(* IEC 61131-3 sources: std_i2980_v2.06_cp053/Source/IMM/ieccontrol/ServiceNet, 6 files *)

(* ---- FBSendData.pu ---- *)
(*
@h    ! WARNING !
@h    The Kemro K2 system (including software) only meets category B according to EN 954-1,
@h    thus it is not intended for usage in safety-relevant control applications in the field
@h    of personal safety (e.g. emergency stop).
@h    To implement potentially necessary safety-relevant control tasks, always use additional
@h    external safety devices that are intended for the particular purpose, and meet the necessary
@h    functional safety.
@h    For further information see EN 954-1 (EN ISO 13849-1) and/or the K2-x00 user manual, chapter
@h    "CE conformity, directives and standards".

function block for sending data according to ServiceNet protocol to ServiceNet Server.
sends connection data and connection status on raising edge on execute
sends connection status information if status changed, but at least once each 30 seconds (keep alive).

ATTENTION: when changing content of send buffer:
-> ensure that maximum length does not exceed 255 characters per buffer element when concating strings,
   otherwise characters are truncated which will lead to an invalid object beeing sent.
-> ensure to CONCAT sClear String (255 x blank) at the end of each buffer-array element
   (to delete string data stored previously on that buffer element in case the new string is shorter)
-> a string data element started in a buffer element (character ") must be closed in the same buffer element
   because at the end of each 255 character buffer element a zero byte (string terminator) is inserted automatically.
   a zero byte is not allowed in string elements!
   therefore the maximum length of a string that can be sent is 255 - 2 = 253 characters.
*)

IMPORT_OVER_LISTFILE
 GET_RUNTIME
, ABVersionManager
, tyRequestFrom
, tsMachineInfo
, tnConnectionStatus
, tySBuf
, KNETWORK_TcpSend
, TON

END_IMPORT

FUNCTION_BLOCK FBSendData #DUMMY_EDIT_BLOCK

VAR_INPUT
 Execute : BOOL (* sends all data on raising edge, when TRUE: connection status is sent on valuechange and after 30 seconds elapsed without valuechange *);
 TcpHdl : REFERENCE (* handle of an established TCP connection to use for sending data *);
 VersionServiceNetClient : DINT (* ServiceNet protocol version used by client *);
END_VAR

VAR_IN_OUT
 abVersionInfo : ABVersionManager (* block for reading versioninfos and systemname *);
END_VAR

VAR_OUTPUT
 Error : BOOL (* indicates a send error *);
END_VAR

SYSTEM_VAR
 sv_RequestFrom : tyRequestFrom;
 sv_sTextMessage : STRING(255);
 sv_iRequestFromIdx : DINT;
 sv_iCpuId : LINT;
 sv_MachineInformation : tsMachineInfo;
 sv_ConnectionStatus : tnConnectionStatus;
 sv_iRemoteVisType : DINT;
END_VAR

VAR
 Buf : tySBuf (* send buffer *);
 fbTCPSend : KNETWORK_TcpSend (* block for sending data  *);
 bSendConnectionData : BOOL (* indicates all data should be sent *);
 bSendStatusOnly : BOOL (* indicates only status should be sent *);
 bExecuteOld : BOOL (* flag stores Execute state in previous cycle for detecting edges *);
 ts : TIME (* debug: timestamp start *);
 td : TIME (* debug: duration *);
 fbTonKeepAlive : TON (* keep alive timer *);
 iConnectionState : DINT (* integer value of sv_ConnectionState *);
 connectionStatusOld : tnConnectionStatus (* connection state in previous cycle - to detect state changed *);
 iSendBytes : UDINT (* number of bytes to send *);
 sByteLen : STRING(16) (* length information about data object to be sent to ServiceNet server *);
 sTmpString : STRING(63) (* helper string  *);
 sKVSVersion : STRING(63);
END_VAR

VAR CONSTANT
 sClear : STRING(255) := '                                                                                                                                                                                                                                                               ' (* string with 255 blanks (0x20) *);
END_VAR
#BEGIN_EDIT_BLOCK
(**************************************** WARNING ********************************************
 *** The KEBA Kemro K2 System including software is not intended for safety control tasks! ***
 ***                       For further information see Comment tab!                        ***
 *********************************************************************************************)

// keep alive message timer, start on raising edge of Execute input
fbTonKeepAlive(Execute, T#30s);

// data to send if keep alive timer elapsed or connection status changed
bSendStatusOnly := fbTonKeepAlive.Q OR (sv_ConnectionStatus <> connectionStatusOld);

// initialize TCP send block on raising edge
IF (Execute AND (NOT bExecuteOld)) THEN
    fbTCPSend(Execute := FALSE, TcpHdl := TcpHdl);
END_IF;

IF (Execute) THEN
   // send all connection data on raising edget of Execute flag
   bSendConnectionData := (NOT bExecuteOld);

   // send data?
   IF (bSendStatusOnly OR bSendConnectionData) THEN
       // reset keep alive timer
       fbTonKeepAlive(IN := FALSE);

       // timestamp for performance measurement
       ts := GET_RUNTIME();

       connectionStatusOld := sv_ConnectionStatus;

       // connection status to integer
       CASE (connectionStatusOld) OF
            nDisconnected:
                iConnectionState := 0;

            nConnecting:
                iConnectionState := 1;

            nRequestPending:
                iConnectionState := 2;

            nServiceAccepted:
                iConnectionState := 3;

            nServiceAccessRequest:
                iConnectionState := 4;

           nServiceActive:
                iConnectionState := 5;
       ELSE
            Error := TRUE;
       END_CASE;

       // length of data object to send
       IF (bSendConnectionData) THEN
            // length with all connection data
            iSendBytes := 256 * 8; // integer with number of bytes to send for tcp send block
            sByteLen := "SJSN0100000007F8"; // 8 byte protocol info, ASCII coded 4 byte hexadecimal with number of bytes
       ELSE
            // length of connection status object
            iSendBytes := 256;
            sByteLen := "00000100";
       END_IF;

       // fill sendbuffer:
       // 8 byte length information followed by JSON object containing payload
       // according to ServiceNet Server protocol
       Buf[0] := CONCAT(sByteLen, '{"ConnectionState":', DINT_TO_STRING(iConnectionState));

       IF (bSendConnectionData) THEN
           // send all connection data
           Buf[0] := CONCAT(Buf[0],
                            ',"ConnectionData":{"UserData":{"CustomerName":"',
                            sv_MachineInformation.sCustomerName,
                            '"',
                            sClear
                           );

           Buf[1] := CONCAT(',"MachineName":"', sv_MachineInformation.sMachineName,
                            '","CountryCode":"', sv_MachineInformation.sCountryCode,
                            '"',
                            sClear
                           );

           Buf[2] := CONCAT(',"LicenseKey":"', sv_MachineInformation.sLicenseKey,
                            '","Request.Name":"', sv_RequestFrom[sv_iRequestFromIdx].sName,
                            '","Request.SkypeName":"', sv_RequestFrom[sv_iRequestFromIdx].sSkypeName,
                            '"',
                            sClear
                           );

           Buf[3] := CONCAT(',"Request.EMail":"', sv_RequestFrom[sv_iRequestFromIdx].sEmail,
                            '@', sv_RequestFrom[sv_iRequestFromIdx].sEmail2,
                            '","Request.Phone":"', sv_RequestFrom[sv_iRequestFromIdx].sPhoneNumber,
                            '","TxtMsg":',
                            sClear
                           );

           // limit textmessage to 253
           IF (LEN(sv_sTextMessage) > 253) THEN
              sv_sTextMessage := LEFT(sv_sTextMessage, 253);
           END_IF;
           Buf[4] := CONCAT('"', sv_sTextMessage, '"', sClear);

           sTmpString := abVersionInfo.fGetSystemName();
           Buf[5] := CONCAT('},"AddInfo":{"RemoteVisType":',
                            DINT_TO_STRING(sv_iRemoteVisType),
                            ', "VersionServiceNetClient":',
                            DINT_TO_STRING(VersionServiceNetClient),
                            '},"ControllerInfo":{"SystemName":"',
                            sTmpString,
                            '","CPUSerial":"',
                            LINT_TO_STRING(sv_iCpuId), '"',
                            sClear);

           sTmpString := abVersionInfo.fGetIECVersion();
           Buf[6] := CONCAT(',"KePlast.IEC":"', sTmpString, '"');

           sTmpString := abVersionInfo.fGetKVBVersion();
           Buf[6] := CONCAT(Buf[6], ',"KePlast.HMI.KVB":"', sTmpString, '"');

           IF (sKVSVersion = '') THEN
               sKVSVersion := abVersionInfo.fReadKVSVersion();
           END_IF;
           Buf[6] := CONCAT(Buf[6], ',"KePlast.HMI.KVS":"', sKVSVersion, '"', sClear);

           sTmpString := abVersionInfo.fGetFirmwareVersion();
           Buf[7] := CONCAT(',"Firmware":"', sTmpString, '"}}}', sClear);
       ELSE
           // send connection state only
           Buf[0] := CONCAT(Buf[0], '}', sClear);
       END_IF;

       // send data
       fbTCPSend(TRUE, TcpHdl, iSendBytes, Buf);

       // calculate runtime
       td := GET_RUNTIME() - ts;

       // set error flag if any error on send
       Error := Error OR fbTCPSend.Error;

       bSendStatusOnly := FALSE;
   END_IF;
END_IF;

// clear outputs and local status vars if Execute false
IF (NOT Execute) THEN
    Error := FALSE;
    bSendStatusOnly := FALSE;
END_IF;

bExecuteOld := Execute;

;#END_EDIT_BLOCK END_FUNCTION_BLOCK

#END_OF_IEC_PART

@Puma @IecEditor 6 121 @Pou 25
@@@BEG_Comment@@@
@h    ! WARNING !
@h    The Kemro K2 system (including software) only meets category B according to EN 954-1,
@h    thus it is not intended for usage in safety-relevant control applications in the field
@h    of personal safety (e.g. emergency stop).
@h    To implement potentially necessary safety-relevant control tasks, always use additional
@h    external safety devices that are intended for the particular purpose, and meet the necessary
@h    functional safety.
@h    For further information see EN 954-1 (EN ISO 13849-1) and/or the K2-x00 user manual, chapter
@h    "CE conformity, directives and standards".

function block for sending data according to ServiceNet protocol to ServiceNet Server.
sends connection data and connection status on raising edge on execute
sends connection status information if status changed, but at least once each 30 seconds (keep alive).

ATTENTION: when changing content of send buffer:
-> ensure that maximum length does not exceed 255 characters per buffer element when concating strings,
   otherwise characters are truncated which will lead to an invalid object beeing sent.
-> ensure to CONCAT sClear String (255 x blank) at the end of each buffer-array element
   (to delete string data stored previously on that buffer element in case the new string is shorter)
-> a string data element started in a buffer element (character ") must be closed in the same buffer element
   because at the end of each 255 character buffer element a zero byte (string terminator) is inserted automatically.
   a zero byte is not allowed in string elements!
   therefore the maximum length of a string that can be sent is 255 - 2 = 253 characters.
@@@END_Comment@@@

@BEG_Contents

@BEG_Func
@RT(17)FuncTreeContainer
1
@Var @RT(11)GET_RUNTIME @RT(0) @T @T @DERIVED 0 @F @RT(22)KEBA_STANDARD_FUNCTION @F
@T
@BEG_Attrib
0 @RT(0) @RT(0)
@END_Attrib
1 1 @F @F @F @F

@END_Func

@BEG_Const
@RT(18)ConstTreeContainer
0
@END_Const

@BEG_Export

@BEG_Kind
@FUNCTION_BLOCK @RT(10)FBSendData @STRUCTURED_TEXT
@RT(0) @RT(0) @RT(0)
@END_Kind

@BEG_Dcl
@RT(16)DclTreeContainer
27
@Var @RT(7)Execute @RT(0) @T @F @DT @RT(4)BOOL @RT(0) @T @T @BASIC 0 @F
@F @F
@T
@BEG_Attrib
3 @RT(0) @RT(132)sends all data on raising edge, when TRUE: connection status is sent on valuechange and after 30 seconds elapsed without valuechange @RT(0)
@END_Attrib
1 1 @F @F @F @F

@Var @RT(6)TcpHdl @RT(0) @T @F @DT @RT(9)REFERENCE @RT(0) @T @T @BASIC 0 @F
@F @F
@T
@BEG_Attrib
3 @RT(0) @RT(63)handle of an established TCP connection to use for sending data @RT(0)
@END_Attrib
1 1 @F @F @F @F

@Var @RT(23)VersionServiceNetClient @RT(0) @T @F @DT @RT(4)DINT @RT(0) @T @T @BASIC 0 @F
@F @F
@T
@BEG_Attrib
3 @RT(0) @RT(42)ServiceNet protocol version used by client @RT(0)
@END_Attrib
1 1 @F @F @F @F

@Var @RT(13)abVersionInfo @RT(0) @T @T @DERIVED 0 @T @T @DT @RT(16)ABVersionManager @RT(0) @T @T @UNKNOWN 0 @F
@F @F
@T
@BEG_Attrib
3 @RT(0) @RT(45)block for reading versioninfos and systemname @RT(0)
@END_Attrib
1 2 @F @F @F @F

@Var @RT(5)Error @RT(0) @T @F @DT @RT(4)BOOL @RT(0) @T @T @BASIC 0 @F
@F @F
@T
@BEG_Attrib
3 @RT(0) @RT(22)indicates a send error @RT(0)
@END_Attrib
1 3 @F @F @F @F

@Var @RT(14)sv_RequestFrom @RT(0) @T @T @DERIVED 0 @T @T @DT @RT(13)tyRequestFrom @RT(0) @T @T @UNKNOWN 0 @F
@F @F
@T
@BEG_Attrib
3 @RT(0) @RT(0) @RT(0)
@END_Attrib
1 8 @F @F @F @F

@Var @RT(15)sv_sTextMessage @RT(0) @T @F @DT @RT(11)STRING(255) @RT(0) @T @T @STRING 0 @F @RT(3)255 @F
@F @F
@T
@BEG_Attrib
3 @RT(0) @RT(0) @RT(0)
@END_Attrib
1 8 @F @F @F @F

@Var @RT(18)sv_iRequestFromIdx @RT(0) @T @F @DT @RT(4)DINT @RT(0) @T @T @BASIC 0 @F
@F @F
@T
@BEG_Attrib
3 @RT(0) @RT(0) @RT(0)
@END_Attrib
1 8 @F @F @F @F

@Var @RT(9)sv_iCpuId @RT(0) @T @F @DT @RT(4)LINT @RT(0) @T @T @BASIC 0 @F
@F @F
@T
@BEG_Attrib
3 @RT(0) @RT(0) @RT(0)
@END_Attrib
1 8 @F @F @F @F

@Var @RT(21)sv_MachineInformation @RT(0) @T @T @DERIVED 0 @T @T @DT @RT(13)tsMachineInfo @RT(0) @T @T @UNKNOWN 0 @F
@F @F
@T
@BEG_Attrib
3 @RT(0) @RT(0) @RT(0)
@END_Attrib
1 8 @F @F @F @F

@Var @RT(19)sv_ConnectionStatus @RT(0) @T @T @DERIVED 0 @T @T @DT @RT(18)tnConnectionStatus @RT(0) @T @T @UNKNOWN 0 @F
@F @F
@T
@BEG_Attrib
3 @RT(0) @RT(0) @RT(0)
@END_Attrib
1 8 @F @F @F @F

@Var @RT(17)sv_iRemoteVisType @RT(0) @T @F @DT @RT(4)DINT @RT(0) @T @T @BASIC 0 @F
@F @F
@T
@BEG_Attrib
3 @RT(0) @RT(0) @RT(0)
@END_Attrib
1 8 @F @F @F @F

@Var @RT(3)Buf @RT(0) @T @T @DERIVED 0 @T @T @DT @RT(6)tySBuf @RT(0) @T @T @UNKNOWN 0 @F
@F @F
@T
@BEG_Attrib
3 @RT(0) @RT(11)send buffer @RT(0)
@END_Attrib
1 0 @F @F @F @F

@Var @RT(9)fbTCPSend @RT(0) @T @T @DERIVED 0 @T @T @DT @RT(16)KNETWORK_TcpSend @RT(0) @T @T @UNKNOWN 0 @F
@F @F
@T
@BEG_Attrib
3 @RT(0) @RT(23)block for sending data  @RT(0)
@END_Attrib
1 0 @F @F @F @F

@Var @RT(19)bSendConnectionData @RT(0) @T @F @DT @RT(4)BOOL @RT(0) @T @T @BASIC 0 @F
@F @F
@T
@BEG_Attrib
3 @RT(0) @RT(33)indicates all data should be sent @RT(0)
@END_Attrib
1 0 @F @F @F @F

@Var @RT(15)bSendStatusOnly @RT(0) @T @F @DT @RT(4)BOOL @RT(0) @T @T @BASIC 0 @F
@F @F
@T
@BEG_Attrib
3 @RT(0) @RT(36)indicates only status should be sent @RT(0)
@END_Attrib
1 0 @F @F @F @F

@Var @RT(11)bExecuteOld @RT(0) @T @F @DT @RT(4)BOOL @RT(0) @T @T @BASIC 0 @F
@F @F
@T
@BEG_Attrib
3 @RT(0) @RT(63)flag stores Execute state in previous cycle for detecting edges @RT(0)
@END_Attrib
1 0 @F @F @F @F

@Var @RT(6)sClear @RT(0) @T @F @DT @RT(11)STRING(255) @RT(0) @T @T @STRING 0 @F @RT(3)255 @F
@F @F
@T
@BEG_Attrib
3 @RT(257)'                                                                                                                                                                                                                                                               ' @RT(29)string with 255 blanks (0x20) @RT(0)
@END_Attrib
1 15 @F @F @F @F

@Var @RT(2)ts @RT(0) @T @F @DT @RT(4)TIME @RT(0) @T @T @BASIC 0 @F
@F @F
@T
@BEG_Attrib
3 @RT(0) @RT(22)debug: timestamp start @RT(0)
@END_Attrib
1 0 @F @F @F @F

@Var @RT(2)td @RT(0) @T @F @DT @RT(4)TIME @RT(0) @T @T @BASIC 0 @F
@F @F
@T
@BEG_Attrib
3 @RT(0) @RT(15)debug: duration @RT(0)
@END_Attrib
1 0 @F @F @F @F

@Var @RT(14)fbTonKeepAlive @RT(0) @T @T @DERIVED 0 @T @T @DT @RT(3)TON @RT(0) @T @T @UNKNOWN 0 @F
@F @F
@T
@BEG_Attrib
3 @RT(0) @RT(16)keep alive timer @RT(0)
@END_Attrib
1 0 @F @F @F @F

@Var @RT(16)iConnectionState @RT(0) @T @F @DT @RT(4)DINT @RT(0) @T @T @BASIC 0 @F
@F @F
@T
@BEG_Attrib
3 @RT(0) @RT(35)integer value of sv_ConnectionState @RT(0)
@END_Attrib
1 0 @F @F @F @F

@Var @RT(19)connectionStatusOld @RT(0) @T @T @DERIVED 0 @T @T @DT @RT(18)tnConnectionStatus @RT(0) @T @T @UNKNOWN 0 @F
@F @F
@T
@BEG_Attrib
3 @RT(0) @RT(60)connection state in previous cycle - to detect state changed @RT(0)
@END_Attrib
1 0 @F @F @F @F

@Var @RT(10)iSendBytes @RT(0) @T @F @DT @RT(5)UDINT @RT(0) @T @T @BASIC 0 @F
@F @F
@T
@BEG_Attrib
3 @RT(0) @RT(23)number of bytes to send @RT(0)
@END_Attrib
1 0 @F @F @F @F

@Var @RT(8)sByteLen @RT(0) @T @F @DT @RT(10)STRING(16) @RT(0) @T @T @STRING 0 @F @RT(2)16 @F
@F @F
@T
@BEG_Attrib
3 @RT(0) @RT(68)length information about data object to be sent to ServiceNet server @RT(0)
@END_Attrib
1 0 @F @F @F @F

@Var @RT(10)sTmpString @RT(0) @T @F @DT @RT(10)STRING(63) @RT(0) @T @T @STRING 0 @F @RT(2)63 @F
@F @F
@T
@BEG_Attrib
3 @RT(0) @RT(14)helper string  @RT(0)
@END_Attrib
1 0 @F @F @F @F

@Var @RT(11)sKVSVersion @RT(0) @T @F @DT @RT(10)STRING(63) @RT(0) @T @T @STRING 0 @F @RT(2)63 @F
@F @F
@T
@BEG_Attrib
3 @RT(0) @RT(0) @RT(0)
@END_Attrib
1 0 @F @F @F @F

@END_Dcl

@END_Export

@BEG_Body
@TL(158)
(**************************************** WARNING ********************************************
 *** The KEBA Kemro K2 System including software is not intended for safety control tasks! ***
 ***                       For further information see Comment tab!                        ***
 *********************************************************************************************)

// keep alive message timer, start on raising edge of Execute input
fbTonKeepAlive(Execute, T#30s);

// data to send if keep alive timer elapsed or connection status changed
bSendStatusOnly := fbTonKeepAlive.Q OR (sv_ConnectionStatus <> connectionStatusOld);

// initialize TCP send block on raising edge
IF (Execute AND (NOT bExecuteOld)) THEN
    fbTCPSend(Execute := FALSE, TcpHdl := TcpHdl);
END_IF;

IF (Execute) THEN
   // send all connection data on raising edget of Execute flag
   bSendConnectionData := (NOT bExecuteOld);

   // send data?
   IF (bSendStatusOnly OR bSendConnectionData) THEN
       // reset keep alive timer
       fbTonKeepAlive(IN := FALSE);

       // timestamp for performance measurement
       ts := GET_RUNTIME();

       connectionStatusOld := sv_ConnectionStatus;

       // connection status to integer
       CASE (connectionStatusOld) OF
            nDisconnected:
                iConnectionState := 0;

            nConnecting:
                iConnectionState := 1;

            nRequestPending:
                iConnectionState := 2;

            nServiceAccepted:
                iConnectionState := 3;

            nServiceAccessRequest:
                iConnectionState := 4;

           nServiceActive:
                iConnectionState := 5;
       ELSE
            Error := TRUE;
       END_CASE;

       // length of data object to send
       IF (bSendConnectionData) THEN
            // length with all connection data
            iSendBytes := 256 * 8; // integer with number of bytes to send for tcp send block
            sByteLen := "SJSN0100000007F8"; // 8 byte protocol info, ASCII coded 4 byte hexadecimal with number of bytes
       ELSE
            // length of connection status object
            iSendBytes := 256;
            sByteLen := "00000100";
       END_IF;

       // fill sendbuffer:
       // 8 byte length information followed by JSON object containing payload
       // according to ServiceNet Server protocol
       Buf[0] := CONCAT(sByteLen, '{"ConnectionState":', DINT_TO_STRING(iConnectionState));

       IF (bSendConnectionData) THEN
           // send all connection data
           Buf[0] := CONCAT(Buf[0],
                            ',"ConnectionData":{"UserData":{"CustomerName":"',
                            sv_MachineInformation.sCustomerName,
                            '"',
                            sClear
                           );

           Buf[1] := CONCAT(',"MachineName":"', sv_MachineInformation.sMachineName,
                            '","CountryCode":"', sv_MachineInformation.sCountryCode,
                            '"',
                            sClear
                           );

           Buf[2] := CONCAT(',"LicenseKey":"', sv_MachineInformation.sLicenseKey,
                            '","Request.Name":"', sv_RequestFrom[sv_iRequestFromIdx].sName,
                            '","Request.SkypeName":"', sv_RequestFrom[sv_iRequestFromIdx].sSkypeName,
                            '"',
                            sClear
                           );

           Buf[3] := CONCAT(',"Request.EMail":"', sv_RequestFrom[sv_iRequestFromIdx].sEmail,
                            '@', sv_RequestFrom[sv_iRequestFromIdx].sEmail2,
                            '","Request.Phone":"', sv_RequestFrom[sv_iRequestFromIdx].sPhoneNumber,
                            '","TxtMsg":',
                            sClear
                           );

           // limit textmessage to 253
           IF (LEN(sv_sTextMessage) > 253) THEN
              sv_sTextMessage := LEFT(sv_sTextMessage, 253);
           END_IF;
           Buf[4] := CONCAT('"', sv_sTextMessage, '"', sClear);

           sTmpString := abVersionInfo.fGetSystemName();
           Buf[5] := CONCAT('},"AddInfo":{"RemoteVisType":',
                            DINT_TO_STRING(sv_iRemoteVisType),
                            ', "VersionServiceNetClient":',
                            DINT_TO_STRING(VersionServiceNetClient),
                            '},"ControllerInfo":{"SystemName":"',
                            sTmpString,
                            '","CPUSerial":"',
                            LINT_TO_STRING(sv_iCpuId), '"',
                            sClear);

           sTmpString := abVersionInfo.fGetIECVersion();
           Buf[6] := CONCAT(',"KePlast.IEC":"', sTmpString, '"');

           sTmpString := abVersionInfo.fGetKVBVersion();
           Buf[6] := CONCAT(Buf[6], ',"KePlast.HMI.KVB":"', sTmpString, '"');

           IF (sKVSVersion = '') THEN
               sKVSVersion := abVersionInfo.fReadKVSVersion();
           END_IF;
           Buf[6] := CONCAT(Buf[6], ',"KePlast.HMI.KVS":"', sKVSVersion, '"', sClear);

           sTmpString := abVersionInfo.fGetFirmwareVersion();
           Buf[7] := CONCAT(',"Firmware":"', sTmpString, '"}}}', sClear);
       ELSE
           // send connection state only
           Buf[0] := CONCAT(Buf[0], '}', sClear);
       END_IF;

       // send data
       fbTCPSend(TRUE, TcpHdl, iSendBytes, Buf);

       // calculate runtime
       td := GET_RUNTIME() - ts;

       // set error flag if any error on send
       Error := Error OR fbTCPSend.Error;

       bSendStatusOnly := FALSE;
   END_IF;
END_IF;

// clear outputs and local status vars if Execute false
IF (NOT Execute) THEN
    Error := FALSE;
    bSendStatusOnly := FALSE;
END_IF;

bExecuteOld := Execute;

@END_Body

@END_Contents

(* ---- FBSNNetworkConfig.pu ---- *)
(*
@h    ! WARNING !
@h    The Kemro K2 system (including software) only meets category B according to EN 954-1,
@h    thus it is not intended for usage in safety-relevant control applications in the field
@h    of personal safety (e.g. emergency stop).
@h    To implement potentially necessary safety-relevant control tasks, always use additional
@h    external safety devices that are intended for the particular purpose, and meet the necessary
@h    functional safety.
@h    For further information see EN 954-1 (EN ISO 13849-1) and/or the K2-x00 user manual, chapter
@h    "CE conformity, directives and standards".

used to change network configuration temporary to values defined in sv_SNNetworkConfig
*)

IMPORT_OVER_LISTFILE
 KNetworkConfigGet
, KNetworkConfigSet
, tsNetworkCfg

END_IMPORT

FUNCTION_BLOCK FBSNNetworkConfig #DUMMY_EDIT_BLOCK

VAR_INPUT
 UseServiceNetConfig : BOOL;
END_VAR

VAR_OUTPUT
 Error : BOOL;
END_VAR

SYSTEM_VAR
 sv_SNNetworkConfig : tsNetworkCfg (* network config to use when connecting to servicenet *);
END_VAR

VAR_TEMP
 ret : BOOL;
END_VAR

VAR
 originalNetworkConfig : tsNetworkCfg (* network config to use when connecting to servicenet *);
 bServiceNetConfig : BOOL;
END_VAR
#BEGIN_EDIT_BLOCK
(**************************************** WARNING ********************************************
 *** The KEBA Kemro K2 System including software is not intended for safety control tasks! ***
 ***                       For further information see Comment tab!                        ***
 *********************************************************************************************)

IF (sv_SNNetworkConfig.sIP = "") THEN
    // no network config change required
    Error := FALSE;
    RETURN;
END_IF;

IF (bServiceNetConfig <> UseServiceNetConfig) THEN
   IF (UseServiceNetConfig) THEN
       // initial read of actual network config
       IF (originalNetworkConfig.sIP = "") THEN
           ret := KNetworkConfigGet(0,
                                    originalNetworkConfig.sIP,
                                    originalNetworkConfig.sSubnetMask,
                                    originalNetworkConfig.sGateway);
       ELSE
           ret := TRUE;
       END_IF;

       IF (ret) THEN
           // set network config servicenet
           ret := KNetworkConfigSet(0,
                                    sv_SNNetworkConfig.sIP,
                                    sv_SNNetworkConfig.sSubnetMask,
                                    sv_SNNetworkConfig.sGateway);
       END_IF;
   ELSE
       // set network config original
       IF (originalNetworkConfig.sIP <> "0.0.0.0") THEN
           ret := KNetworkConfigSet(0,
                                originalNetworkConfig.sIP,
                                originalNetworkConfig.sSubnetMask,
                                originalNetworkConfig.sGateway);
       ELSE
           ret := TRUE;
       END_IF;
   END_IF;
END_IF;

IF (ret) THEN
   bServiceNetConfig := UseServiceNetConfig;
   Error := FALSE;
ELSE
   Error := TRUE;
END_IF;

;#END_EDIT_BLOCK END_FUNCTION_BLOCK

#END_OF_IEC_PART

@Puma @IecEditor 6 128 @Pou 25
@@@BEG_Comment@@@
@h    ! WARNING !
@h    The Kemro K2 system (including software) only meets category B according to EN 954-1,
@h    thus it is not intended for usage in safety-relevant control applications in the field
@h    of personal safety (e.g. emergency stop).
@h    To implement potentially necessary safety-relevant control tasks, always use additional
@h    external safety devices that are intended for the particular purpose, and meet the necessary
@h    functional safety.
@h    For further information see EN 954-1 (EN ISO 13849-1) and/or the K2-x00 user manual, chapter
@h    "CE conformity, directives and standards".

used to change network configuration temporary to values defined in sv_SNNetworkConfig
@@@END_Comment@@@

@BEG_Contents

@BEG_Func
@RT(17)FuncTreeContainer
2
@Var @RT(17)KNetworkConfigGet @RT(0) @T @T @DERIVED 0 @F @RT(22)KEBA_STANDARD_FUNCTION @F
@T
@BEG_Attrib
0 @RT(0) @RT(0)
@END_Attrib
1 1 @F @F @F @F

@Var @RT(17)KNetworkConfigSet @RT(0) @T @T @DERIVED 0 @F @RT(22)KEBA_STANDARD_FUNCTION @F
@T
@BEG_Attrib
0 @RT(0) @RT(0)
@END_Attrib
1 1 @F @F @F @F

@END_Func

@BEG_Const
@RT(18)ConstTreeContainer
0
@END_Const

@BEG_Export

@BEG_Kind
@FUNCTION_BLOCK @RT(17)FBSNNetworkConfig @STRUCTURED_TEXT
@RT(0) @RT(0) @RT(0)
@END_Kind

@BEG_Dcl
@RT(16)DclTreeContainer
6
@Var @RT(18)sv_SNNetworkConfig @RT(0) @T @T @DERIVED 0 @T @T @DT @RT(12)tsNetworkCfg @RT(0) @T @T @UNKNOWN 0 @F
@F @F
@T
@BEG_Attrib
3 @RT(0) @RT(51)network config to use when connecting to servicenet @RT(0)
@END_Attrib
1 8 @F @F @F @F

@Var @RT(21)originalNetworkConfig @RT(0) @T @T @DERIVED 0 @T @T @DT @RT(12)tsNetworkCfg @RT(0) @T @T @UNKNOWN 0 @F
@F @F
@T
@BEG_Attrib
3 @RT(0) @RT(51)network config to use when connecting to servicenet @RT(0)
@END_Attrib
1 0 @F @F @F @F

@Var @RT(19)UseServiceNetConfig @RT(0) @T @F @DT @RT(4)BOOL @RT(0) @T @T @BASIC 0 @F
@F @F
@T
@BEG_Attrib
3 @RT(0) @RT(0) @RT(0)
@END_Attrib
1 1 @F @F @F @F

@Var @RT(17)bServiceNetConfig @RT(0) @T @F @DT @RT(4)BOOL @RT(0) @T @T @BASIC 0 @F
@F @F
@T
@BEG_Attrib
3 @RT(0) @RT(0) @RT(0)
@END_Attrib
1 0 @F @F @F @F

@Var @RT(3)ret @RT(0) @T @F @DT @RT(4)BOOL @RT(0) @T @T @BASIC 0 @F
@F @F
@T
@BEG_Attrib
3 @RT(0) @RT(0) @RT(0)
@END_Attrib
1 4 @F @F @F @F

@Var @RT(5)Error @RT(0) @T @F @DT @RT(4)BOOL @RT(0) @T @T @BASIC 0 @F
@F @F
@T
@BEG_Attrib
3 @RT(0) @RT(0) @RT(0)
@END_Attrib
1 3 @F @F @F @F

@END_Dcl

@END_Export

@BEG_Body
@TL(51)
(**************************************** WARNING ********************************************
 *** The KEBA Kemro K2 System including software is not intended for safety control tasks! ***
 ***                       For further information see Comment tab!                        ***
 *********************************************************************************************)

IF (sv_SNNetworkConfig.sIP = "") THEN
    // no network config change required
    Error := FALSE;
    RETURN;
END_IF;

IF (bServiceNetConfig <> UseServiceNetConfig) THEN
   IF (UseServiceNetConfig) THEN
       // initial read of actual network config
       IF (originalNetworkConfig.sIP = "") THEN
           ret := KNetworkConfigGet(0,
                                    originalNetworkConfig.sIP,
                                    originalNetworkConfig.sSubnetMask,
                                    originalNetworkConfig.sGateway);
       ELSE
           ret := TRUE;
       END_IF;

       IF (ret) THEN
           // set network config servicenet
           ret := KNetworkConfigSet(0,
                                    sv_SNNetworkConfig.sIP,
                                    sv_SNNetworkConfig.sSubnetMask,
                                    sv_SNNetworkConfig.sGateway);
       END_IF;
   ELSE
       // set network config original
       IF (originalNetworkConfig.sIP <> "0.0.0.0") THEN
           ret := KNetworkConfigSet(0,
                                originalNetworkConfig.sIP,
                                originalNetworkConfig.sSubnetMask,
                                originalNetworkConfig.sGateway);
       ELSE
           ret := TRUE;
       END_IF;
   END_IF;
END_IF;

IF (ret) THEN
   bServiceNetConfig := UseServiceNetConfig;
   Error := FALSE;
ELSE
   Error := TRUE;
END_IF;

@END_Body

@END_Contents

(* ---- ABModemCfg.pu ---- *)
(*
@h    ! WARNING !
@h    The Kemro K2 system (including software) only meets category B according to EN 954-1,
@h    thus it is not intended for usage in safety-relevant control applications in the field
@h    of personal safety (e.g. emergency stop).
@h    To implement potentially necessary safety-relevant control tasks, always use additional
@h    external safety devices that are intended for the particular purpose, and meet the necessary
@h    functional safety.
@h    For further information see EN 954-1 (EN ISO 13849-1) and/or the K2-x00 user manual, chapter
@h    "CE conformity, directives and standards".

The Algorithm sends the SIM Configuration (pin, apn, user, password) to an MB connect modem.

*)

IMPORT_OVER_LISTFILE
 START_PROCESS_ALGORITHM
, STOP_PROCESS_ALGORITHM
, SET_ALARM
, RESET_ALARM
, cHttp_PortNumber
, tsSimInfo
, tsNetworkCfg
, KNETWORK_TcpInit
, KNETWORK_TcpSend
, KNETWORK_TcpReceive
, KNETWORK_Event
, FBSNNetworkConfig

END_IMPORT

ALGORITHM_BLOCK ABModemCfg #DUMMY_EDIT_BLOCK

SYSTEM_VAR
 sv_bDownloadSIMInfo : BOOL;
 sv_iDownloadSIMInfoErrorCode : DINT;
 sv_SIMInfo : tsSimInfo;
 sv_bConnect : BOOL;
 sv_SNNetworkConfig : tsNetworkCfg (* network config to use when connecting to servicenet *);
END_VAR

SYSTEM_OBJECT
 TaskSlow : TASK;
 erDownloadSimInfoFailed : ALARM;
END_OBJECT

VAR
 iModemCfgState : DINT := 0;
END_VAR

POSTUPDATE_ALGORITHM pModemCfg ON TaskSlow WITH sv_bDownloadSIMInfo

VAR
 dummy : DINT;
END_VAR
#BEGIN_EDIT_BLOCK
IF (sv_bDownloadSIMInfo) THEN
    IF (sv_bConnect) THEN
        // not allowed, download sim info in progress
        dummy := Print("Modem configuration: servicenet connected -> download could not be startet !");
        sv_iDownloadSIMInfoErrorCode := 100;
        sv_bDownloadSIMInfo := FALSE;
    ELSE
        sv_iDownloadSIMInfoErrorCode := 0;
        iModemCfgState := 0;
        START_PROCESS_ALGORITHM(paDoModemCfg);
    END_IF;
END_IF;

;#END_EDIT_BLOCK END_ALGORITHM

PROCESS_ALGORITHM paDoModemCfg ON TaskSlow

VAR
 fbKNETWORK_TcpInit : KNETWORK_TcpInit;
 fbKNETWORK_TcpSend : KNETWORK_TcpSend;
 fbKNETWORK_TcpReceive : KNETWORK_TcpReceive;
 evKNETWORK : KNETWORK_Event;
 bError : BOOL := FALSE;
 bDone : BOOL := FALSE;
 dErrorID : DWORD;
 pTcpHdl : REFERENCE;
 sSendData : STRING(255);
 sReceiveData : STRING(255);
 sActCommand : STRING(63);
 sCommandSetsim1 : STRING(63) := 'setsim1';
 sCommandApply : STRING(63) := 'apply';
 dBytesReceived : UDINT := 0;
 iCommandParamResult : INT;
 iCommandResult : INT;
 bReconnect : BOOL;
 iModemCfgStateOld : DINT;
 iHelp : INT;
 iSendDataLen : UDINT;
 iReplyWaitCnt : INT := 0;
 Dummy : DINT;
 iTimeoutCnt : DINT := 0;
 fbSNNetConfig : FBSNNetworkConfig;
END_VAR
#BEGIN_EDIT_BLOCK
CASE iModemCfgState OF

    0:  // Initialize
        iModemCfgStateOld := 0;
        sActCommand := sCommandSetsim1;
        bReconnect := FALSE;
        iTimeoutCnt := 0;
        iReplyWaitCnt := 0;
        iModemCfgState := 1;
        RESET_ALARM(Name := erDownloadSimInfoFailed);
        fbSNNetConfig(UseServiceNetConfig := TRUE);
        IF (fbSNNetConfig.Error) THEN
            Dummy := Print("Modem configuration: error when setting temp network config");
            sv_iDownloadSIMInfoErrorCode := 110;
            iModemCfgState := 10;    // error -> disconnect and abort
        END_IF;

    1:  // Connect to modem
        Dummy := Print("Modem configuration: Try to connect to %s port %d", sv_SNNetworkConfig.sGateway, cHttp_PortNumber);
        fbKNETWORK_TcpInit (Execute := TRUE, RemoteIP := sv_SNNetworkConfig.sGateway, RemotePort := cHttp_PortNumber, NotificationEvent := evKNETWORK,
                            Done => bDone, Error => bError, ErrorID => dErrorID, TcpHdl => pTcpHdl);

        IF (bDone = TRUE) THEN
            Dummy := Print("Modem configuration: Connection successfully established");
            iModemCfgState := 3;    // send request to modem
        END_IF;

        IF (bError = TRUE) THEN
            Dummy := Print("Modem configuration: ERROR connecting to %s port %d", sv_SNNetworkConfig.sGateway, cHttp_PortNumber);
            sv_iDownloadSIMInfoErrorCode := DWORD_TO_DINT(dErrorID);
            iModemCfgState := 10;    // error -> abort
        END_IF;

    2:   // Disconnect from modem
        Dummy := Print("Modem configuration: Close connection %s port %d", sv_SNNetworkConfig.sGateway, cHttp_PortNumber);
        fbKNETWORK_TcpInit (Execute := FALSE, Done => bDone, Error => bError, ErrorID => dErrorID);

        IF (bDone = TRUE) THEN
            Dummy := Print("Modem configuration: Connection successfully closed");
        END_IF;
        IF (bError = TRUE) THEN
            Dummy := Print("Modem configuration: ERROR closing connection");
            sv_iDownloadSIMInfoErrorCode := DWORD_TO_DINT(dErrorID);
        END_IF;

        IF (bDone = TRUE) OR (bError = TRUE) THEN
            IF (bReconnect = TRUE) THEN
                bReconnect := FALSE;
                iModemCfgState := 1;    // Reconnect
            ELSE
                iModemCfgState := 10;   // done -> abort
            END_IF;
        END_IF;

    3:  // Create request string
        sSendData := "";

        IF (sActCommand = sCommandSetsim1) THEN
            sSendData := "GET /cgi-bin/cfg.sh?action=setsim1&pin=";
            sSendData := CONCAT(sSendData, sv_SIMInfo.sPIN);

            sSendData := CONCAT(sSendData, "&apn=");
            sSendData := CONCAT(sSendData, sv_SIMInfo.sAPN);

            sSendData := CONCAT(sSendData, "&user=");
            IF (LEN(sv_SIMInfo.sUserName) = 0) THEN
                sSendData := CONCAT(sSendData, "noUser");
            ELSE
                sSendData := CONCAT(sSendData, sv_SIMInfo.sUserName);
            END_IF;

            sSendData := CONCAT(sSendData, "&pass=");
            IF (LEN(sv_SIMInfo.sPassword) = 0) THEN
                sSendData := CONCAT(sSendData, "noPass");
            ELSE
                sSendData := CONCAT(sSendData, sv_SIMInfo.sPassword);
            END_IF;
        END_IF;
        IF (sActCommand = sCommandApply) THEN
            sSendData := "GET /cgi-bin/cfg.sh?action=apply";
        END_IF;

        sSendData := CONCAT(sSendData, " HTTP/1.1$N");
        sSendData := CONCAT(sSendData, "Host: ");
        sSendData := CONCAT(sSendData, sv_SNNetworkConfig.sGateway);
        sSendData := CONCAT(sSendData, "$N");
        sSendData := CONCAT(sSendData, "Authorization: Basic YWRtaW46");    // password: admin
        sSendData := CONCAT(sSendData, "$N$N");

        iModemCfgState := 4;

    4:  // Send request to modem
        iSendDataLen := LEN(sSendData);
        Dummy := Print("Modem configuration: Send request (len %u): %s", iSendDataLen, sSendData);

        fbKNETWORK_TcpSend(Execute := TRUE, TcpHdl := pTcpHdl, DataLen := iSendDataLen, Data := sSendData,
                           Done => bDone, Error => bError, ErrorID => dErrorID);

        IF (bDone = TRUE) THEN
            iModemCfgState := 6;    // wait for request reply
        END_IF;

        IF (bError = TRUE) THEN
            sv_iDownloadSIMInfoErrorCode := DWORD_TO_DINT(dErrorID);
            iModemCfgState := 2;    // error -> disconnect and abort
        END_IF;

    6:  // wait for request reply
        // reduction of trace outputs
        IF (MOD(iReplyWaitCnt, 10) = 0) THEN
            Dummy := Print("Modem configuration: waiting for data ...");
        END_IF;

        iReplyWaitCnt := iReplyWaitCnt + 1;
        sReceiveData := "";
        fbKNETWORK_TcpReceive (Execute := TRUE, TcpHdl := pTcpHdl, DataBufferLen := 255, DataBuffer := sReceiveData,
                               Done => bDone, Error => bError, ErrorID => dErrorID, BytesReceived => dBytesReceived);

        IF (bDone = TRUE) THEN
            // data received -> analyze status
            IF (dBytesReceived > 0) THEN
                Dummy := Print("Modem configuration: received data: %s", sReceiveData);

                iCommandParamResult := 0;       // command parameter result
                iCommandResult      := 0;       // command result
                iHelp := FIND(sReceiveData, sActCommand);

                IF (iHelp > 0) THEN
                    iHelp := iHelp + LEN(sActCommand) + 1;

                    iCommandParamResult := STRING_TO_INT(MID(sReceiveData, 1, iHelp));
                    iCommandResult      := STRING_TO_INT(MID(sReceiveData, 1, iHelp + 2));
                END_IF;

                IF (iCommandParamResult = 1) AND (iCommandResult = 1) THEN
                    // successfully done
                    Dummy := Print("Modem configuration: Request successfully finished");
                    IF (sActCommand = sCommandSetsim1) THEN
                        // next command: apply (disconnect and reconnect to modem necessary)
                        sActCommand := sCommandApply;
                        bReconnect := TRUE;
                    END_IF;
                ELSE
                    // error occured
                    IF (iCommandParamResult = 0) THEN
                        Dummy := Print("Modem configuration: request parameter error");
                        sv_iDownloadSIMInfoErrorCode := 101;
                    END_IF;
                    IF (iCommandResult = 0) THEN
                        Dummy := Print("Modem configuration: request command error");
                        sv_iDownloadSIMInfoErrorCode := 102;
                    END_IF;
                END_IF;
                iModemCfgState := 2;
            END_IF;
        END_IF;

        IF (bError = TRUE) THEN
            sv_iDownloadSIMInfoErrorCode := DWORD_TO_DINT(dErrorID);
            iModemCfgState := 2;    // error -> disconnect and abort
        END_IF;

    10: // ready - done
        fbSNNetConfig(UseServiceNetConfig := FALSE);
        IF (fbSNNetConfig.Error) THEN
            Dummy := Print("Modem configuration: error when reset temp network config");
            sv_iDownloadSIMInfoErrorCode := 111;
            iModemCfgState := 10;    // error -> disconnect and abort
        END_IF;

        sv_bDownloadSIMInfo := FALSE;
        IF (sv_iDownloadSIMInfoErrorCode <> 0) THEN
            iHelp := DINT_TO_INT(sv_iDownloadSIMInfoErrorCode);
            SET_ALARM(Name := erDownloadSimInfoFailed, Param1 := iHelp);
        END_IF;
        STOP_PROCESS_ALGORITHM();

ELSE
    Dummy := Print("Modem configuration: ERROR - invalid state %i", iModemCfgState);
    sv_iDownloadSIMInfoErrorCode := 110;
    iModemCfgState := 10;
END_CASE;

IF (iModemCfgState <> iModemCfgStateOld) THEN
    iModemCfgStateOld := iModemCfgState;
    iTimeoutCnt := 0;
END_IF;

// check for timeout (if iModemCfgState does not change for a several time -> timeout)
IF (iTimeoutCnt > 200) THEN
    Dummy := Print("Modem configuration: Timeout occured");

    iTimeoutCnt := 0;
    sv_iDownloadSIMInfoErrorCode := 105;
    iModemCfgState := 2;
ELSE
    iTimeoutCnt := iTimeoutCnt + 1;
END_IF;

;#END_EDIT_BLOCK END_ALGORITHM

END_ALGORITHM_BLOCK

#END_OF_IEC_PART

@Puma @IecEditor 6 127 @Pou 25
@@@BEG_Comment@@@
@h    ! WARNING !
@h    The Kemro K2 system (including software) only meets category B according to EN 954-1,
@h    thus it is not intended for usage in safety-relevant control applications in the field
@h    of personal safety (e.g. emergency stop).
@h    To implement potentially necessary safety-relevant control tasks, always use additional
@h    external safety devices that are intended for the particular purpose, and meet the necessary
@h    functional safety.
@h    For further information see EN 954-1 (EN ISO 13849-1) and/or the K2-x00 user manual, chapter
@h    "CE conformity, directives and standards".

The Algorithm sends the SIM Configuration (pin, apn, user, password) to an MB connect modem.

@@@END_Comment@@@

@BEG_Contents

@BEG_Func
@RT(17)FuncTreeContainer
4
@Var @RT(23)START_PROCESS_ALGORITHM @RT(0) @T @T @DERIVED 0 @F @RT(23)KEBA_STANDARD_PROCEDURE @F
@T
@BEG_Attrib
0 @RT(0) @RT(0)
@END_Attrib
1 1 @F @F @F @F

@Var @RT(22)STOP_PROCESS_ALGORITHM @RT(0) @T @T @DERIVED 0 @F @RT(23)KEBA_STANDARD_PROCEDURE @F
@T
@BEG_Attrib
0 @RT(0) @RT(0)
@END_Attrib
1 1 @F @F @F @F

@Var @RT(9)SET_ALARM @RT(0) @T @T @DERIVED 0 @F @RT(23)KEBA_STANDARD_PROCEDURE @F
@T
@BEG_Attrib
0 @RT(0) @RT(0)
@END_Attrib
1 1 @F @F @F @F

@Var @RT(11)RESET_ALARM @RT(0) @T @T @DERIVED 0 @F @RT(23)KEBA_STANDARD_PROCEDURE @F
@T
@BEG_Attrib
0 @RT(0) @RT(0)
@END_Attrib
1 1 @F @F @F @F

@END_Func

@BEG_Const
@RT(18)ConstTreeContainer
1
@Var @RT(16)cHttp_PortNumber @RT(0) @T @F @DT @RT(4)WORD @RT(0) @T @T @BASIC 0 @F
@F @F
@T
@BEG_Attrib
0 @RT(2)80 @RT(40)port number for HTTP connection to modem
@END_Attrib
1 1 @F @F @F @F

@END_Const

@BEG_Export

@BEG_Kind
@ALGORITHM_BLOCK @RT(10)ABModemCfg @STRUCTURED_TEXT
@RT(0) @RT(0) @RT(0)
@END_Kind

@BEG_Dcl
@RT(16)DclTreeContainer
8
@Var @RT(8)TaskSlow @RT(0) @T @T @RENAMED 0 @T @T @DT @RT(4)TASK @RT(0) @T @T @BASIC 0 @F
@F @F
@T
@BEG_Attrib
3 @RT(0) @RT(0) @RT(0)
@END_Attrib
1 7 @F @F @F @F

@Var @RT(19)sv_bDownloadSIMInfo @RT(0) @T @F @DT @RT(4)BOOL @RT(0) @T @T @BASIC 0 @F
@F @F
@T
@BEG_Attrib
3 @RT(0) @RT(0) @RT(0)
@END_Attrib
1 8 @F @F @F @F

@Var @RT(28)sv_iDownloadSIMInfoErrorCode @RT(0) @T @F @DT @RT(4)DINT @RT(0) @T @T @BASIC 0 @F
@F @F
@T
@BEG_Attrib
3 @RT(0) @RT(0) @RT(0)
@END_Attrib
1 8 @F @F @F @F

@Var @RT(10)sv_SIMInfo @RT(0) @T @T @DERIVED 0 @T @T @DT @RT(9)tsSimInfo @RT(0) @T @T @UNKNOWN 0 @F
@F @F
@T
@BEG_Attrib
3 @RT(0) @RT(0) @RT(0)
@END_Attrib
1 8 @F @F @F @F

@Var @RT(14)iModemCfgState @RT(0) @T @F @DT @RT(4)DINT @RT(0) @T @T @BASIC 0 @F
@F @F
@T
@BEG_Attrib
3 @RT(1)0 @RT(0) @RT(0)
@END_Attrib
1 0 @F @F @F @F

@Var @RT(23)erDownloadSimInfoFailed @RT(0) @T @F @DT @RT(5)ALARM @RT(0) @T @T @BASIC 0 @F
@F @F
@T
@BEG_Attrib
3 @RT(0) @RT(0) @RT(0)
@END_Attrib
1 7 @F @F @F @F

@Var @RT(11)sv_bConnect @RT(0) @T @F @DT @RT(4)BOOL @RT(0) @T @T @BASIC 0 @F
@F @F
@T
@BEG_Attrib
3 @RT(0) @RT(0) @RT(0)
@END_Attrib
1 8 @F @F @F @F

@Var @RT(18)sv_SNNetworkConfig @RT(0) @T @T @DERIVED 0 @T @T @DT @RT(12)tsNetworkCfg @RT(0) @T @T @UNKNOWN 0 @F
@F @F
@T
@BEG_Attrib
3 @RT(0) @RT(51)network config to use when connecting to servicenet @RT(0)
@END_Attrib
1 8 @F @F @F @F

@END_Dcl

@END_Export

@BEG_Body

2

@BEG_Export

@BEG_Algo
@POSTUPDATE_ALGORITHM @RT(9)pModemCfg @STRUCTURED_TEXT
@RT(0) @RT(19)sv_bDownloadSIMInfo @RT(8)TaskSlow @F @F
@END_Algo

@BEG_Dcl
@RT(16)DclTreeContainer
1
@Var @RT(5)dummy @RT(0) @T @F @DT @RT(4)DINT @RT(0) @T @T @BASIC 0 @F
@F @F
@T
@BEG_Attrib
3 @RT(0) @RT(0) @RT(0)
@END_Attrib
1 0 @F @F @F @F

@END_Dcl

@END_Export

@BEG_Export

@BEG_Algo
@PROCESS_ALGORITHM @RT(12)paDoModemCfg @STRUCTURED_TEXT
@RT(0) @RT(0) @RT(8)TaskSlow @F @F
@END_Algo

@BEG_Dcl
@RT(16)DclTreeContainer
24
@Var @RT(18)fbKNETWORK_TcpInit @RT(0) @T @T @DERIVED 0 @T @T @DT @RT(16)KNETWORK_TcpInit @RT(0) @T @T @UNKNOWN 0 @F
@F @F
@T
@BEG_Attrib
3 @RT(0) @RT(0) @RT(0)
@END_Attrib
1 0 @F @F @F @F

@Var @RT(18)fbKNETWORK_TcpSend @RT(0) @T @T @DERIVED 0 @T @T @DT @RT(16)KNETWORK_TcpSend @RT(0) @T @T @UNKNOWN 0 @F
@F @F
@T
@BEG_Attrib
3 @RT(0) @RT(0) @RT(0)
@END_Attrib
1 0 @F @F @F @F

@Var @RT(21)fbKNETWORK_TcpReceive @RT(0) @T @T @DERIVED 0 @T @T @DT @RT(19)KNETWORK_TcpReceive @RT(0) @T @T @UNKNOWN 0 @F
@F @F
@T
@BEG_Attrib
3 @RT(0) @RT(0) @RT(0)
@END_Attrib
1 0 @F @F @F @F

@Var @RT(10)evKNETWORK @RT(0) @T @T @DERIVED 0 @T @T @DT @RT(14)KNETWORK_Event @RT(0) @T @T @UNKNOWN 0 @F
@F @F
@T
@BEG_Attrib
3 @RT(0) @RT(0) @RT(0)
@END_Attrib
1 0 @F @F @F @F

@Var @RT(6)bError @RT(0) @T @F @DT @RT(4)BOOL @RT(0) @T @T @BASIC 0 @F
@F @F
@T
@BEG_Attrib
3 @RT(5)FALSE @RT(0) @RT(0)
@END_Attrib
1 0 @F @F @F @F

@Var @RT(5)bDone @RT(0) @T @F @DT @RT(4)BOOL @RT(0) @T @T @BASIC 0 @F
@F @F
@T
@BEG_Attrib
3 @RT(5)FALSE @RT(0) @RT(0)
@END_Attrib
1 0 @F @F @F @F

@Var @RT(8)dErrorID @RT(0) @T @F @DT @RT(5)DWORD @RT(0) @T @T @BASIC 0 @F
@F @F
@T
@BEG_Attrib
3 @RT(0) @RT(0) @RT(0)
@END_Attrib
1 0 @F @F @F @F

@Var @RT(7)pTcpHdl @RT(0) @T @F @DT @RT(9)REFERENCE @RT(0) @T @T @BASIC 0 @F
@F @F
@T
@BEG_Attrib
3 @RT(0) @RT(0) @RT(0)
@END_Attrib
1 0 @F @F @F @F

@Var @RT(9)sSendData @RT(0) @T @F @DT @RT(11)STRING(255) @RT(0) @T @T @STRING 0 @F @RT(3)255 @F
@F @F
@T
@BEG_Attrib
3 @RT(0) @RT(0) @RT(0)
@END_Attrib
1 0 @F @F @F @F

@Var @RT(12)sReceiveData @RT(0) @T @F @DT @RT(11)STRING(255) @RT(0) @T @T @STRING 0 @F @RT(3)255 @F
@F @F
@T
@BEG_Attrib
3 @RT(0) @RT(0) @RT(0)
@END_Attrib
1 0 @F @F @F @F

@Var @RT(11)sActCommand @RT(0) @T @F @DT @RT(10)STRING(63) @RT(0) @T @T @STRING 0 @F @RT(2)63 @F
@F @F
@T
@BEG_Attrib
3 @RT(0) @RT(0) @RT(0)
@END_Attrib
1 0 @F @F @F @F

@Var @RT(15)sCommandSetsim1 @RT(0) @T @F @DT @RT(10)STRING(63) @RT(0) @T @T @STRING 0 @F @RT(2)63 @F
@F @F
@T
@BEG_Attrib
3 @RT(9)'setsim1' @RT(0) @RT(0)
@END_Attrib
1 0 @F @F @F @F

@Var @RT(13)sCommandApply @RT(0) @T @F @DT @RT(10)STRING(63) @RT(0) @T @T @STRING 0 @F @RT(2)63 @F
@F @F
@T
@BEG_Attrib
3 @RT(7)'apply' @RT(0) @RT(0)
@END_Attrib
1 0 @F @F @F @F

@Var @RT(14)dBytesReceived @RT(0) @T @F @DT @RT(5)UDINT @RT(0) @T @T @BASIC 0 @F
@F @F
@T
@BEG_Attrib
3 @RT(1)0 @RT(0) @RT(0)
@END_Attrib
1 0 @F @F @F @F

@Var @RT(19)iCommandParamResult @RT(0) @T @F @DT @RT(3)INT @RT(0) @T @T @BASIC 0 @F
@F @F
@T
@BEG_Attrib
3 @RT(0) @RT(0) @RT(0)
@END_Attrib
1 0 @F @F @F @F

@Var @RT(14)iCommandResult @RT(0) @T @F @DT @RT(3)INT @RT(0) @T @T @BASIC 0 @F
@F @F
@T
@BEG_Attrib
3 @RT(0) @RT(0) @RT(0)
@END_Attrib
1 0 @F @F @F @F

@Var @RT(10)bReconnect @RT(0) @T @F @DT @RT(4)BOOL @RT(0) @T @T @BASIC 0 @F
@F @F
@T
@BEG_Attrib
3 @RT(0) @RT(0) @RT(0)
@END_Attrib
1 0 @F @F @F @F

@Var @RT(17)iModemCfgStateOld @RT(0) @T @F @DT @RT(4)DINT @RT(0) @T @T @BASIC 0 @F
@F @F
@T
@BEG_Attrib
3 @RT(0) @RT(0) @RT(0)
@END_Attrib
1 0 @F @F @F @F

@Var @RT(5)iHelp @RT(0) @T @F @DT @RT(3)INT @RT(0) @T @T @BASIC 0 @F
@F @F
@T
@BEG_Attrib
3 @RT(0) @RT(0) @RT(0)
@END_Attrib
1 0 @F @F @F @F

@Var @RT(12)iSendDataLen @RT(0) @T @F @DT @RT(5)UDINT @RT(0) @T @T @BASIC 0 @F
@F @F
@T
@BEG_Attrib
3 @RT(0) @RT(0) @RT(0)
@END_Attrib
1 0 @F @F @F @F

@Var @RT(13)iReplyWaitCnt @RT(0) @T @F @DT @RT(3)INT @RT(0) @T @T @BASIC 0 @F
@F @F
@T
@BEG_Attrib
3 @RT(1)0 @RT(0) @RT(0)
@END_Attrib
1 0 @F @F @F @F

@Var @RT(5)Dummy @RT(0) @T @F @DT @RT(4)DINT @RT(0) @T @T @BASIC 0 @F
@F @F
@T
@BEG_Attrib
3 @RT(0) @RT(0) @RT(0)
@END_Attrib
1 0 @F @F @F @F

@Var @RT(11)iTimeoutCnt @RT(0) @T @F @DT @RT(4)DINT @RT(0) @T @T @BASIC 0 @F
@F @F
@T
@BEG_Attrib
3 @RT(1)0 @RT(0) @RT(0)
@END_Attrib
1 0 @F @F @F @F

@Var @RT(13)fbSNNetConfig @RT(0) @T @T @DERIVED 0 @T @T @DT @RT(17)FBSNNetworkConfig @RT(0) @T @T @UNKNOWN 0 @F
@F @F
@T
@BEG_Attrib
3 @RT(0) @RT(0) @RT(0)
@END_Attrib
1 0 @F @F @F @F

@END_Dcl

@END_Export

@BEG_Body
@TL(14)
IF (sv_bDownloadSIMInfo) THEN
    IF (sv_bConnect) THEN
        // not allowed, download sim info in progress
        dummy := Print("Modem configuration: servicenet connected -> download could not be startet !");
        sv_iDownloadSIMInfoErrorCode := 100;
        sv_bDownloadSIMInfo := FALSE;
    ELSE
        sv_iDownloadSIMInfoErrorCode := 0;
        iModemCfgState := 0;
        START_PROCESS_ALGORITHM(paDoModemCfg);
    END_IF;
END_IF;

@END_Body

@@@BEG_Comment@@@
@TL(0)

@@@END_Comment@@@

@BEG_Body
@TL(199)
CASE iModemCfgState OF

    0:  // Initialize
        iModemCfgStateOld := 0;
        sActCommand := sCommandSetsim1;
        bReconnect := FALSE;
        iTimeoutCnt := 0;
        iReplyWaitCnt := 0;
        iModemCfgState := 1;
        RESET_ALARM(Name := erDownloadSimInfoFailed);
        fbSNNetConfig(UseServiceNetConfig := TRUE);
        IF (fbSNNetConfig.Error) THEN
            Dummy := Print("Modem configuration: error when setting temp network config");
            sv_iDownloadSIMInfoErrorCode := 110;
            iModemCfgState := 10;    // error -> disconnect and abort
        END_IF;

    1:  // Connect to modem
        Dummy := Print("Modem configuration: Try to connect to %s port %d", sv_SNNetworkConfig.sGateway, cHttp_PortNumber);
        fbKNETWORK_TcpInit (Execute := TRUE, RemoteIP := sv_SNNetworkConfig.sGateway, RemotePort := cHttp_PortNumber, NotificationEvent := evKNETWORK,
                            Done => bDone, Error => bError, ErrorID => dErrorID, TcpHdl => pTcpHdl);

        IF (bDone = TRUE) THEN
            Dummy := Print("Modem configuration: Connection successfully established");
            iModemCfgState := 3;    // send request to modem
        END_IF;

        IF (bError = TRUE) THEN
            Dummy := Print("Modem configuration: ERROR connecting to %s port %d", sv_SNNetworkConfig.sGateway, cHttp_PortNumber);
            sv_iDownloadSIMInfoErrorCode := DWORD_TO_DINT(dErrorID);
            iModemCfgState := 10;    // error -> abort
        END_IF;

    2:   // Disconnect from modem
        Dummy := Print("Modem configuration: Close connection %s port %d", sv_SNNetworkConfig.sGateway, cHttp_PortNumber);
        fbKNETWORK_TcpInit (Execute := FALSE, Done => bDone, Error => bError, ErrorID => dErrorID);

        IF (bDone = TRUE) THEN
            Dummy := Print("Modem configuration: Connection successfully closed");
        END_IF;
        IF (bError = TRUE) THEN
            Dummy := Print("Modem configuration: ERROR closing connection");
            sv_iDownloadSIMInfoErrorCode := DWORD_TO_DINT(dErrorID);
        END_IF;

        IF (bDone = TRUE) OR (bError = TRUE) THEN
            IF (bReconnect = TRUE) THEN
                bReconnect := FALSE;
                iModemCfgState := 1;    // Reconnect
            ELSE
                iModemCfgState := 10;   // done -> abort
            END_IF;
        END_IF;

    3:  // Create request string
        sSendData := "";

        IF (sActCommand = sCommandSetsim1) THEN
            sSendData := "GET /cgi-bin/cfg.sh?action=setsim1&pin=";
            sSendData := CONCAT(sSendData, sv_SIMInfo.sPIN);

            sSendData := CONCAT(sSendData, "&apn=");
            sSendData := CONCAT(sSendData, sv_SIMInfo.sAPN);

            sSendData := CONCAT(sSendData, "&user=");
            IF (LEN(sv_SIMInfo.sUserName) = 0) THEN
                sSendData := CONCAT(sSendData, "noUser");
            ELSE
                sSendData := CONCAT(sSendData, sv_SIMInfo.sUserName);
            END_IF;

            sSendData := CONCAT(sSendData, "&pass=");
            IF (LEN(sv_SIMInfo.sPassword) = 0) THEN
                sSendData := CONCAT(sSendData, "noPass");
            ELSE
                sSendData := CONCAT(sSendData, sv_SIMInfo.sPassword);
            END_IF;
        END_IF;
        IF (sActCommand = sCommandApply) THEN
            sSendData := "GET /cgi-bin/cfg.sh?action=apply";
        END_IF;

        sSendData := CONCAT(sSendData, " HTTP/1.1$N");
        sSendData := CONCAT(sSendData, "Host: ");
        sSendData := CONCAT(sSendData, sv_SNNetworkConfig.sGateway);
        sSendData := CONCAT(sSendData, "$N");
        sSendData := CONCAT(sSendData, "Authorization: Basic YWRtaW46");    // password: admin
        sSendData := CONCAT(sSendData, "$N$N");

        iModemCfgState := 4;

    4:  // Send request to modem
        iSendDataLen := LEN(sSendData);
        Dummy := Print("Modem configuration: Send request (len %u): %s", iSendDataLen, sSendData);

        fbKNETWORK_TcpSend(Execute := TRUE, TcpHdl := pTcpHdl, DataLen := iSendDataLen, Data := sSendData,
                           Done => bDone, Error => bError, ErrorID => dErrorID);

        IF (bDone = TRUE) THEN
            iModemCfgState := 6;    // wait for request reply
        END_IF;

        IF (bError = TRUE) THEN
            sv_iDownloadSIMInfoErrorCode := DWORD_TO_DINT(dErrorID);
            iModemCfgState := 2;    // error -> disconnect and abort
        END_IF;

    6:  // wait for request reply
        // reduction of trace outputs
        IF (MOD(iReplyWaitCnt, 10) = 0) THEN
            Dummy := Print("Modem configuration: waiting for data ...");
        END_IF;

        iReplyWaitCnt := iReplyWaitCnt + 1;
        sReceiveData := "";
        fbKNETWORK_TcpReceive (Execute := TRUE, TcpHdl := pTcpHdl, DataBufferLen := 255, DataBuffer := sReceiveData,
                               Done => bDone, Error => bError, ErrorID => dErrorID, BytesReceived => dBytesReceived);

        IF (bDone = TRUE) THEN
            // data received -> analyze status
            IF (dBytesReceived > 0) THEN
                Dummy := Print("Modem configuration: received data: %s", sReceiveData);

                iCommandParamResult := 0;       // command parameter result
                iCommandResult      := 0;       // command result
                iHelp := FIND(sReceiveData, sActCommand);

                IF (iHelp > 0) THEN
                    iHelp := iHelp + LEN(sActCommand) + 1;

                    iCommandParamResult := STRING_TO_INT(MID(sReceiveData, 1, iHelp));
                    iCommandResult      := STRING_TO_INT(MID(sReceiveData, 1, iHelp + 2));
                END_IF;

                IF (iCommandParamResult = 1) AND (iCommandResult = 1) THEN
                    // successfully done
                    Dummy := Print("Modem configuration: Request successfully finished");
                    IF (sActCommand = sCommandSetsim1) THEN
                        // next command: apply (disconnect and reconnect to modem necessary)
                        sActCommand := sCommandApply;
                        bReconnect := TRUE;
                    END_IF;
                ELSE
                    // error occured
                    IF (iCommandParamResult = 0) THEN
                        Dummy := Print("Modem configuration: request parameter error");
                        sv_iDownloadSIMInfoErrorCode := 101;
                    END_IF;
                    IF (iCommandResult = 0) THEN
                        Dummy := Print("Modem configuration: request command error");
                        sv_iDownloadSIMInfoErrorCode := 102;
                    END_IF;
                END_IF;
                iModemCfgState := 2;
            END_IF;
        END_IF;

        IF (bError = TRUE) THEN
            sv_iDownloadSIMInfoErrorCode := DWORD_TO_DINT(dErrorID);
            iModemCfgState := 2;    // error -> disconnect and abort
        END_IF;

    10: // ready - done
        fbSNNetConfig(UseServiceNetConfig := FALSE);
        IF (fbSNNetConfig.Error) THEN
            Dummy := Print("Modem configuration: error when reset temp network config");
            sv_iDownloadSIMInfoErrorCode := 111;
            iModemCfgState := 10;    // error -> disconnect and abort
        END_IF;

        sv_bDownloadSIMInfo := FALSE;
        IF (sv_iDownloadSIMInfoErrorCode <> 0) THEN
            iHelp := DINT_TO_INT(sv_iDownloadSIMInfoErrorCode);
            SET_ALARM(Name := erDownloadSimInfoFailed, Param1 := iHelp);
        END_IF;
        STOP_PROCESS_ALGORITHM();

ELSE
    Dummy := Print("Modem configuration: ERROR - invalid state %i", iModemCfgState);
    sv_iDownloadSIMInfoErrorCode := 110;
    iModemCfgState := 10;
END_CASE;

IF (iModemCfgState <> iModemCfgStateOld) THEN
    iModemCfgStateOld := iModemCfgState;
    iTimeoutCnt := 0;
END_IF;

// check for timeout (if iModemCfgState does not change for a several time -> timeout)
IF (iTimeoutCnt > 200) THEN
    Dummy := Print("Modem configuration: Timeout occured");

    iTimeoutCnt := 0;
    sv_iDownloadSIMInfoErrorCode := 105;
    iModemCfgState := 2;
ELSE
    iTimeoutCnt := iTimeoutCnt + 1;
END_IF;

@END_Body

@@@BEG_Comment@@@
@TL(0)

@@@END_Comment@@@
@END_Body

@END_Contents
